(* PLC project v0.6.02_RefactorGateAndTest.project, CODESYS CODESYS V3.5 SP19 Patch 1 *)
(* stored: creationDateTime 2026-07-23T23:39:28.699511, modificationDateTime 2026-07-23T23:39:28.699511 *)

(* ═══════════════════════════════════════════════════════════════ 🔧 ST_BucketCfg — Configuration de la benne (M2) ═══════════════════════════════════════════════════════════════ *)
TYPE ST_BucketCfg : STRUCT
  Config : ST_BucketConfig;  (* 🔧 Offsets Open/Close/Coherence *)
  CfgTimeoutDuration : TIME := TIME#30s0ms;  (* ⏱️ Temps max pour l'ouverture/fermeture *)
  Initialized : BOOL := FALSE;  (* 🚦 flag restauration boot *)
END_STRUCT;
END_TYPE

(* ═══════════════════════════════════════════════════════════════ ⚙️ ST_BucketConfig — Configuration des offsets du benne ─────────────────────────────────────────────────────────────── 📄 Doc métier : DOC/AF/AF_Partie-10_Fonction_Winch/FB_Bucket_v1.0.md §4.A ═══════════════════════════════════════════════════════════════ *)
TYPE ST_BucketConfig : STRUCT
  OffsetOpenM : REAL;  (* Écart M1/M2 en mètres benne ouvert *)
  OffsetCloseM : REAL;  (* Écart M1/M2 en mètres benne fermé *)
  CoherenceLimitM : REAL;  (* Seuil de détection d'incohérence au boot *)
  CloseAnticipationM : REAL := 1;  (* 🆕 2026-08-07 (20) — retour terrain, demande client : inertie mécanique du benne (M2 continue sur sa lancée après coupure StartStop) -- couper la commande EN AVANCE de la cible pour que l'arrêt réel (après coast-down) tombe proche du vrai offset, au lieu de dépasser. Anticipation distincte par sens (fermeture/ouverture ont des inerties différentes selon retour terrain). Coupe la commande de fermeture 1m avant OffsetCloseM *)
  OpenAnticipationM : REAL := 1.3;  (* Coupe la commande d'ouverture 1.3m avant OffsetOpenM *)
END_STRUCT;
END_TYPE

(* ═══════════════════════════════════════════════════════════════ 🌉 FB_CfgPersistBridge_BucketCfg — Pont persistance générique pour ST_BucketCfg ─────────────────────────────────────────────────────────────── 🎯 Voir FB_CfgPersistBridge_SyncCfg.st (Lot 3a) pour la logique de référence — identique, seul le type ST_BucketCfg change. La copie struct-à-struct gère aussi le sous-struct imbriqué Config : ST_BucketConfig automatiquement (pas de traitement spécial nécessaire). ═══════════════════════════════════════════════════════════════ *)
FUNCTION_BLOCK FB_CfgPersistBridge_BucketCfg
  VAR_OUTPUT
    JustRestored : BOOL;
  END_VAR
  VAR_IN_OUT
    Hmi : ST_BucketCfg;  (* 🖥️ ex. GVL_IHM.M2TreuilBenne.Bucket.Cfg *)
    Persist : ST_BucketCfg;  (* 💾 ex. GVL_PERSISTENT._BucketCfgPersist *)
  END_VAR

            

JustRestored := FALSE;
IF NOT Hmi.Initialized THEN
    Hmi := Persist;
    Hmi.Initialized := TRUE;
    JustRestored := TRUE;
ELSE
    Persist := Hmi;
END_IF;

          
END_FUNCTION_BLOCK
